{attribute 'qualified_only'}
{attribute 'strict'}
{attribute 'to_string'}
TYPE E_Location :
(
	pl		:= 1,
	en		:= 2,
	de		:= 3
);
END_TYPE

(* stored: Version 1.1.0.1
   DUT E_Location: Id {7db9a948-9705-0032-2a9c-fe43bf593dc2} *)
